# EPICS substitutions: db/Beckhoff_KL/ecmcKL2032.substitutions
#- Not a slave of its own so no ecmcEcSlave.template
#-file "ecmcEcSlave.template"
#-{
#-  pattern {}
#-          {}
#-}

file "ecmcKL2XXX-chx.template"
{
  pattern {CH_ID, ZNAM,   ONAM,   ZSV,        OSV,        PINI,  DESC                               }
          {1,     "Zero", "One",  "NO_ALARM", "NO_ALARM", 1      "$(HWTYPE): Binary Output $(CH_ID)"}
          {2,     "Zero", "One",  "NO_ALARM", "NO_ALARM", 1      "$(HWTYPE): Binary Output $(CH_ID)"}
}
